{attribute addProperty BoxType "EP1816-1008-0016"}
{attribute addProperty Id "DIG_Inputs_ChannelAT %I*ARRAY[0..1] OF DIG_Inputs_Channel_628B507D128160DIG_Inputs_DeviceAT %I*DIG_Inputs_Device_5061D9393240WcStateAT %I*WcState_F855686C1620InfoDataAT %I*InfoData_BC63D37F80100"}
{attribute addProperty CRC "2157604503"}
{attribute addProperty SizeInBites "256"}
{attribute addProperty SizeInBytes "32"}
TYPE EP1816_7BF0AF86 :
STRUCT
	{attribute addProperty Name "DIG_Inputs_Channel"}
	DIG_Inputs_Channel : ARRAY[0..1] OF DIG_Inputs_Channel_628B507D;
	{attribute addProperty Name "DIG_Inputs_Device"}
	DIG_Inputs_Device : DIG_Inputs_Device_5061D939;
	{attribute addProperty Name "WcState"}
	WcState : WcState_F855686C;
	{attribute addProperty Name "InfoData"}
	InfoData : InfoData_BC63D37F;
END_STRUCT
END_TYPE

(* stored: Version 1.2.0.0, ProductVersion 3.1.4024.9
   DUT EP1816_7BF0AF86: Id {57055f87-dd96-4795-a6bc-8bc0fd056323} *)
